{attribute wpf [Container(Layout.Stack)]}
FUNCTION_BLOCK TcoControlVoltage EXTENDS TcoElements.TcoDi IMPLEMENTS  ITcoControlVoltage

VAR_OUTPUT
END_VAR
VAR
END_VAR

SUPER^(inoSignal:=inoSignal);
IF NOT inoSignal THEN
	Messenger.Warning('<#Control Voltage is Off#>');
END_IF;

PROPERTY IsOff : BOOL
GET
IsOff:=not this^._signal;
END_GET
END_PROPERTY

PROPERTY IsOn : BOOL
GET
IsOn:=this^._signal;
END_GET
END_PROPERTY

END_FUNCTION_BLOCK

(* stored: Version 1.1.0.1
   POU TcoControlVoltage: Id {6eae052e-6975-4886-b1fa-a2c2d83e4578}, SpecialFunc None
   Property IsOff: Id {eab858d0-60f4-40dc-9363-46da2e0a7161}
   Get Get: Id {50982d82-b0fa-4178-a9a5-70ba66579ad1}
   Property IsOn: Id {39a9f696-bc19-4831-b729-71e67e01fe3c}
   Get Get: Id {d740a34f-d907-4a76-b38a-f97b3867714d} *)
